// TIA Portal V16 export
// export: Created 2023-07-30T20:35:42.5971621Z, ExportSetting WithDefaults, DisplayName Totally Integrated Automation Portal, DisplayVersion V16, DisplayName TIA Portal Version Control Interface, DisplayVersion V16, DisplayName TIA Portal Openness, DisplayVersion V16, DisplayName STEP 7 Professional, DisplayVersion V16, DisplayName STEP 7 Safety, DisplayVersion V16, DisplayName WinCC Professional, DisplayVersion V16
DATA_BLOCK "Data"   // DB6
{ S7_Optimized_Access := 'TRUE' }
VERSION : 0.1
// stored: AutoNumber true, DBAccessibleFromOPCUA true, IsOnlyStoredInLoadMemory false, IsRetainMemResEnabled false, IsWriteProtectedInAS false, MemoryReserve 100
   VAR
      send : Array[0..3] of Int;
      recv : Array[0..1] of Int;
   END_VAR
BEGIN
   send[0] := 2;
   send[1] := 6;
   send[2] := 8;
   send[3] := 12;
   recv[0] := 5;
   recv[1] := 7;
END_DATA_BLOCK
